FUNCTION WRITE_PROTECTED_LINT
VAR_INPUT
    Ptr : POINTER TO LINT;
    Value : LINT;
END_VAR

Ptr^ := Value;

END_FUNCTION

(* stored: Version 1.1.0.1, ProductVersion 3.1.4022.18
   POU WRITE_PROTECTED_LINT: Id {da64d6c8-2148-431b-b3a7-81dadf9fdad8}, SpecialFunc None *)
